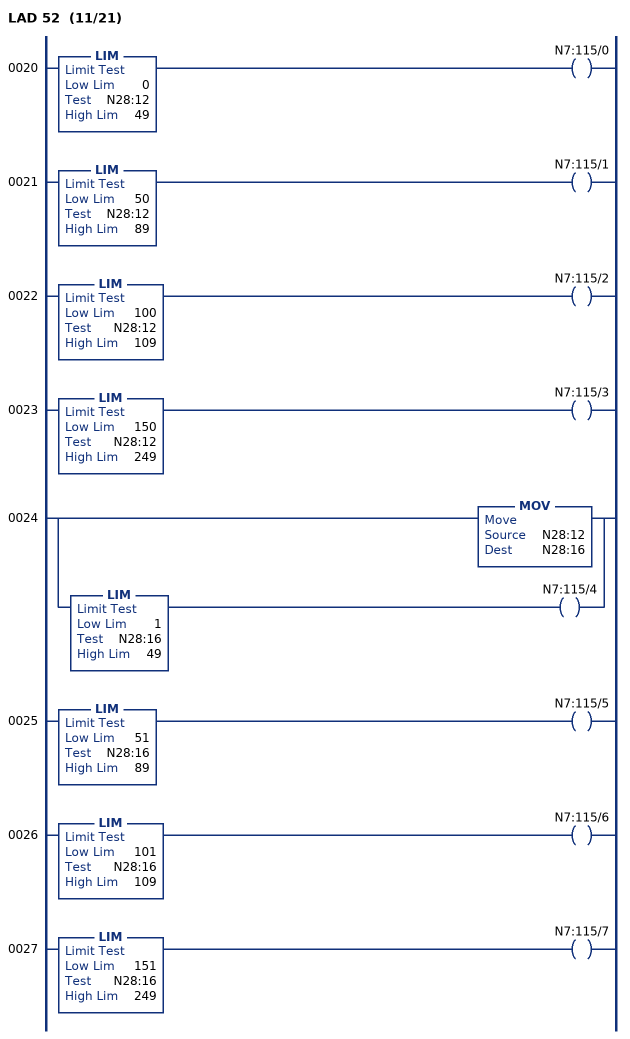
% Rung: 20 %
SOR LIM 0 N28:12 49 OTE N7:115/0 EOR
% Rung: 21 %
SOR LIM 50 N28:12 89 OTE N7:115/1 EOR
% Rung: 22 %
SOR LIM 100 N28:12 109 OTE N7:115/2 EOR
% Rung: 23 %
SOR LIM 150 N28:12 249 OTE N7:115/3 EOR
% Rung: 24 %
SOR BST MOV N28:12 N28:16 NXB LIM 1 N28:16 49 OTE N7:115/4 BND EOR
% Rung: 25 %
SOR LIM 51 N28:16 89 OTE N7:115/5 EOR
% Rung: 26 %
SOR LIM 101 N28:16 109 OTE N7:115/6 EOR
% Rung: 27 %
SOR LIM 151 N28:16 249 OTE N7:115/7 EOR

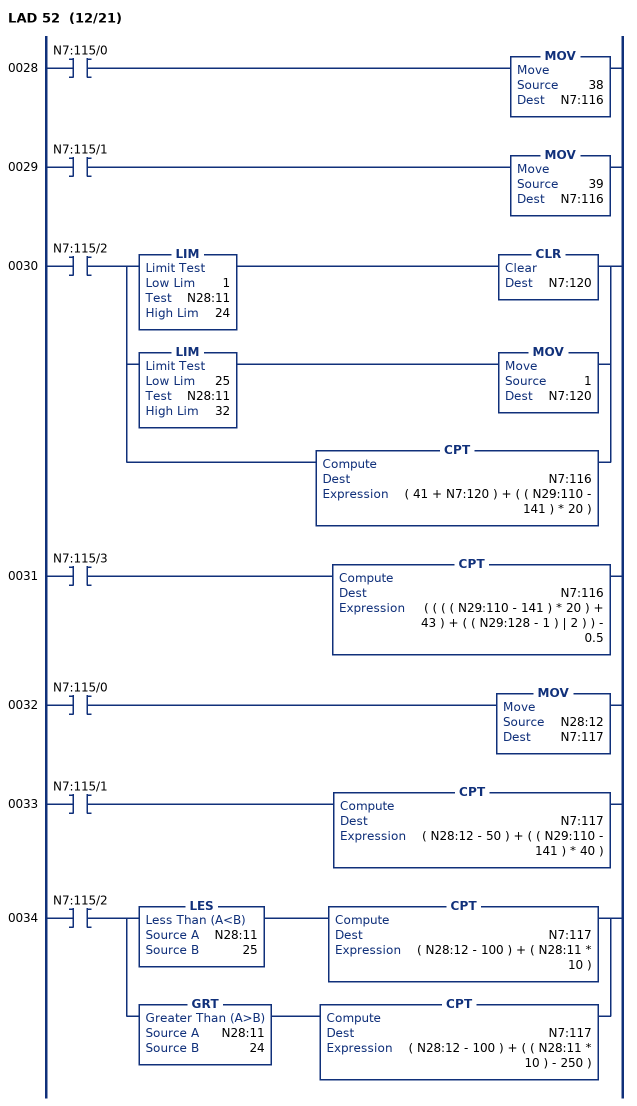
% Rung: 28 %
SOR XIC N7:115/0 MOV 38 N7:116 EOR
% Rung: 29 %
SOR XIC N7:115/1 MOV 39 N7:116 EOR
% Rung: 30 %
SOR XIC N7:115/2 BST LIM 1 N28:11 24 CLR N7:120 NXB LIM 25 N28:11 32 MOV 1 N7:120 NXB CPT N7:116 " ( 41 + N7:120 ) + ( ( N29:110 - 141 ) * 20 ) " BND EOR
% Rung: 31 %
SOR XIC N7:115/3 CPT N7:116 " ( ( ( ( N29:110 - 141 ) * 20 ) + 43 ) + ( ( N29:128 - 1 ) | 2 ) ) - 0.5 " EOR
% Rung: 32 %
SOR XIC N7:115/0 MOV N28:12 N7:117 EOR
% Rung: 33 %
SOR XIC N7:115/1 CPT N7:117 " ( N28:12 - 50 ) + ( ( N29:110 - 141 ) * 40 ) " EOR
% Rung: 34 %
SOR XIC N7:115/2 BST LES N28:11 25 CPT N7:117 " ( N28:12 - 100 ) + ( N28:11 * 10 ) " NXB GRT N28:11 24 CPT N7:117 " ( N28:12 - 100 ) + ( ( N28:11 * 10 ) - 250 ) " BND EOR

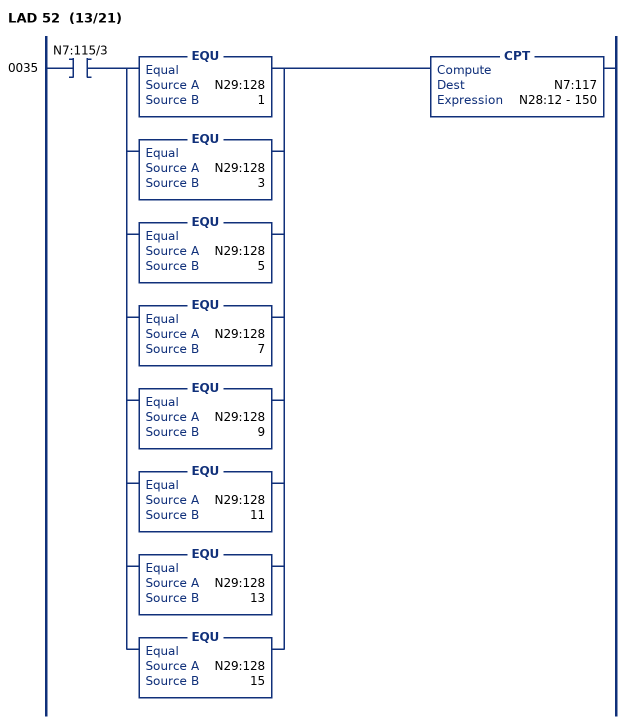
% Rung: 35 %
SOR XIC N7:115/3 BST EQU N29:128 1 NXB EQU N29:128 3 NXB EQU N29:128 5 NXB EQU N29:128 7 NXB EQU N29:128 9 NXB EQU N29:128 11 NXB EQU N29:128 13 NXB EQU N29:128 15 BND CPT N7:117 " N28:12 - 150 " EOR

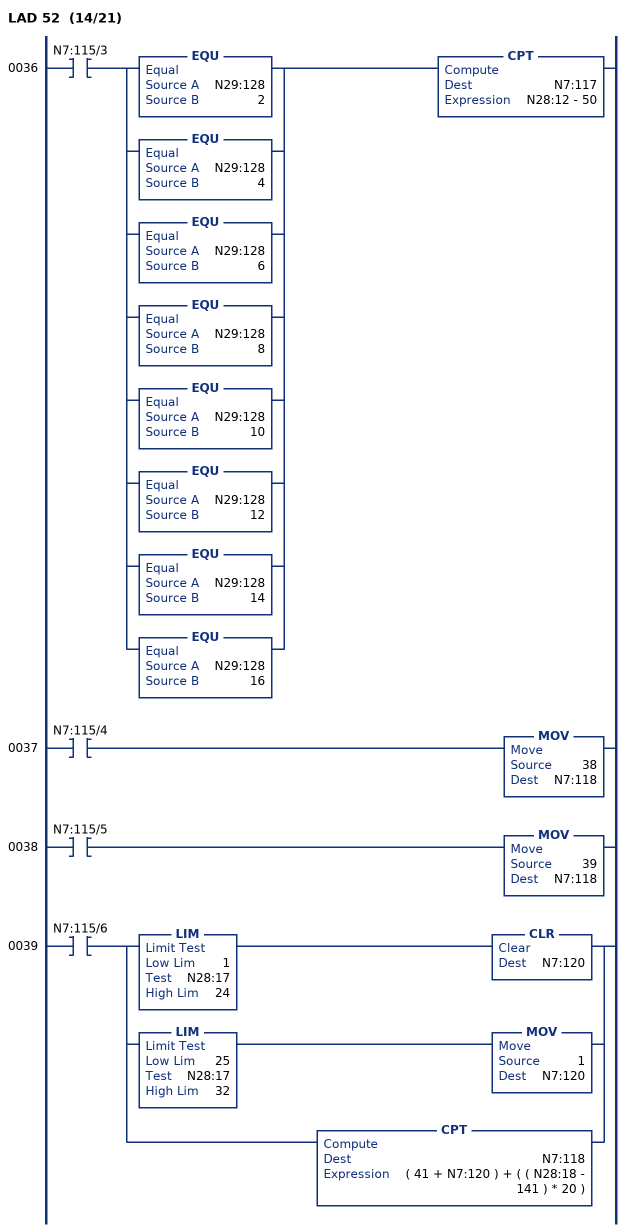
% Rung: 36 %
SOR XIC N7:115/3 BST EQU N29:128 2 NXB EQU N29:128 4 NXB EQU N29:128 6 NXB EQU N29:128 8 NXB EQU N29:128 10 NXB EQU N29:128 12 NXB EQU N29:128 14 NXB EQU N29:128 16 BND CPT N7:117 " N28:12 - 50 " EOR
% Rung: 37 %
SOR XIC N7:115/4 MOV 38 N7:118 EOR
% Rung: 38 %
SOR XIC N7:115/5 MOV 39 N7:118 EOR
% Rung: 39 %
SOR XIC N7:115/6 BST LIM 1 N28:17 24 CLR N7:120 NXB LIM 25 N28:17 32 MOV 1 N7:120 NXB CPT N7:118 " ( 41 + N7:120 ) + ( ( N28:18 - 141 ) * 20 ) " BND EOR

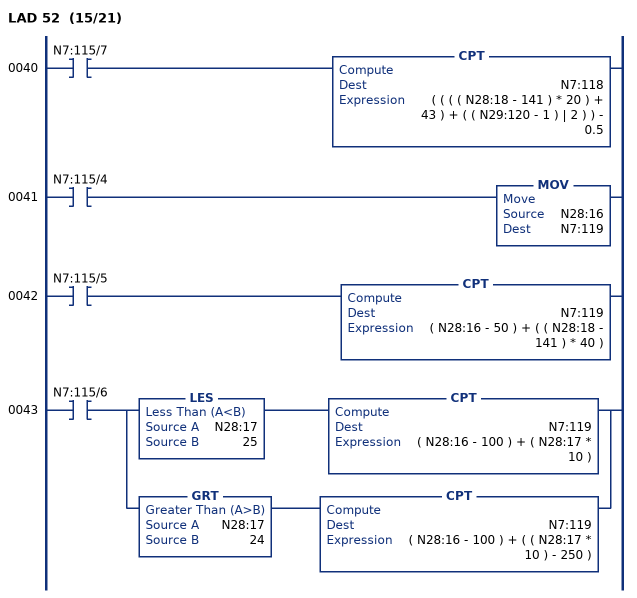
% Rung: 40 %
SOR XIC N7:115/7 CPT N7:118 " ( ( ( ( N28:18 - 141 ) * 20 ) + 43 ) + ( ( N29:120 - 1 ) | 2 ) ) - 0.5 " EOR
% Rung: 41 %
SOR XIC N7:115/4 MOV N28:16 N7:119 EOR
% Rung: 42 %
SOR XIC N7:115/5 CPT N7:119 " ( N28:16 - 50 ) + ( ( N28:18 - 141 ) * 40 ) " EOR
% Rung: 43 %
SOR XIC N7:115/6 BST LES N28:17 25 CPT N7:119 " ( N28:16 - 100 ) + ( N28:17 * 10 ) " NXB GRT N28:17 24 CPT N7:119 " ( N28:16 - 100 ) + ( ( N28:17 * 10 ) - 250 ) " BND EOR

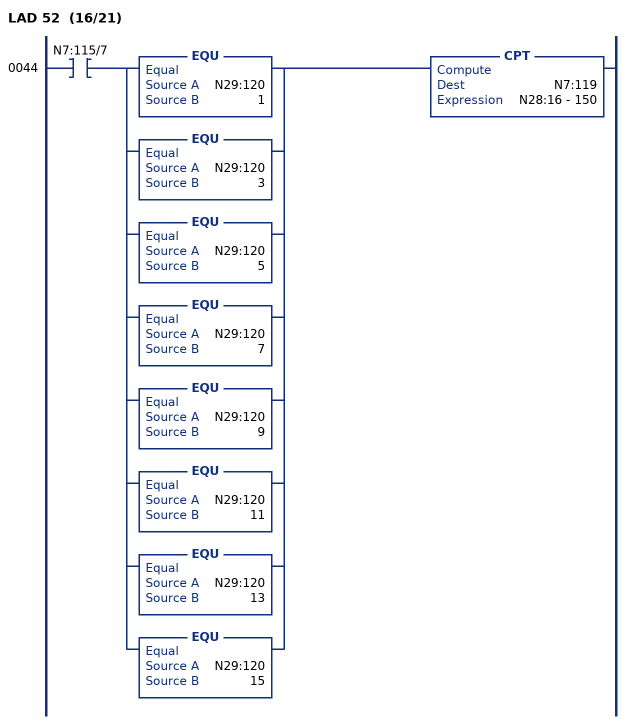
% Rung: 44 %
SOR XIC N7:115/7 BST EQU N29:120 1 NXB EQU N29:120 3 NXB EQU N29:120 5 NXB EQU N29:120 7 NXB EQU N29:120 9 NXB EQU N29:120 11 NXB EQU N29:120 13 NXB EQU N29:120 15 BND CPT N7:119 " N28:16 - 150 " EOR

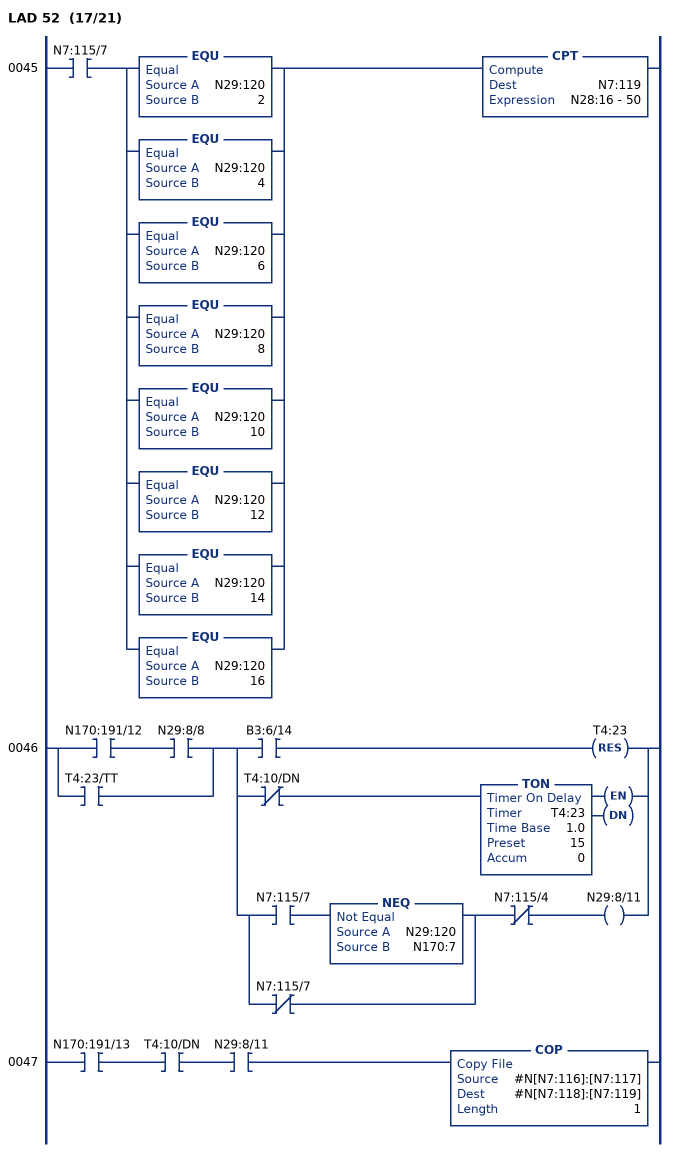
% Rung: 45 %
SOR XIC N7:115/7 BST EQU N29:120 2 NXB EQU N29:120 4 NXB EQU N29:120 6 NXB EQU N29:120 8 NXB EQU N29:120 10 NXB EQU N29:120 12 NXB EQU N29:120 14 NXB EQU N29:120 16 BND CPT N7:119 " N28:16 - 50 " EOR
% Rung: 46 %
SOR BST XIC N170:191/12 XIC N29:8/8 NXB XIC T4:23/TT BND BST XIC B3:6/14 RES T4:23 NXB XIO T4:10/DN TON T4:23 1.0 15 0 NXB BST XIC N7:115/7 NEQ N29:120 N170:7 NXB XIO N7:115/7 BND XIO N7:115/4 OTE N29:8/11 BND EOR
% Rung: 47 %
SOR XIC N170:191/13 XIC T4:10/DN XIC N29:8/11 COP #N[N7:116]:[N7:117] #N[N7:118]:[N7:119] 1 EOR

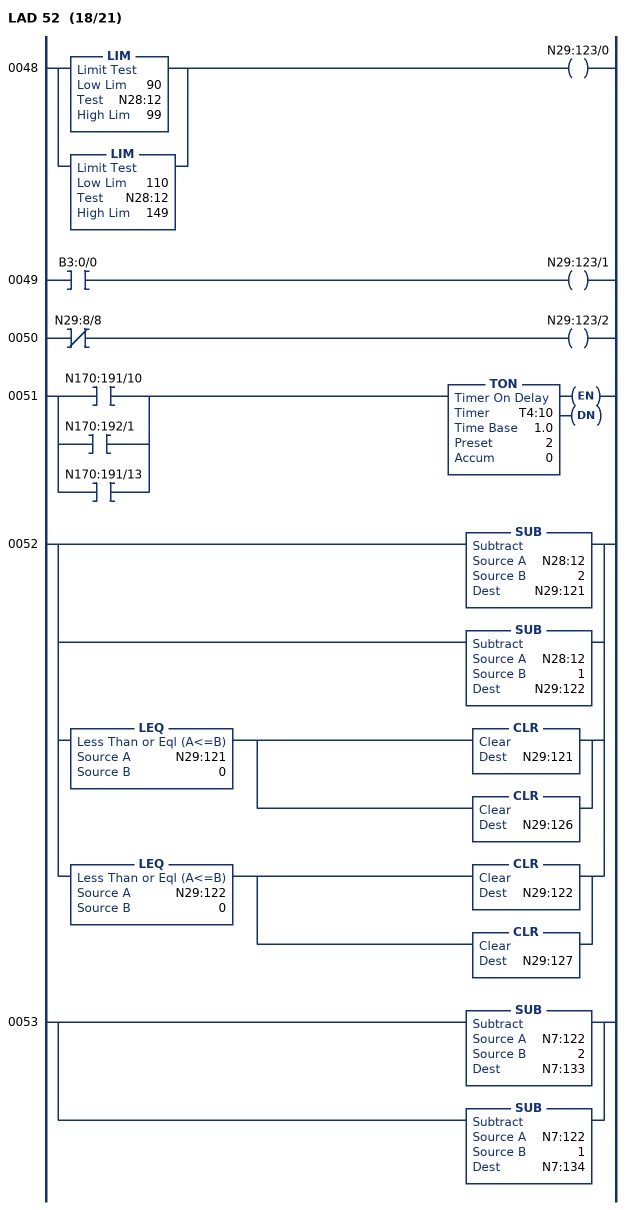
% Rung: 48 %
SOR BST LIM 90 N28:12 99 NXB LIM 110 N28:12 149 BND OTE N29:123/0 EOR
% Rung: 49 %
SOR XIC B3:0/0 OTE N29:123/1 EOR
% Rung: 50 %
SOR XIO N29:8/8 OTE N29:123/2 EOR
% Rung: 51 %
SOR BST XIC N170:191/10 NXB XIC N170:192/1 NXB XIC N170:191/13 BND TON T4:10 1.0 2 0 EOR
% Rung: 52 %
SOR BST SUB N28:12 2 N29:121 NXB SUB N28:12 1 N29:122 NXB LEQ N29:121 0 BST CLR N29:121 NXB CLR N29:126 BND NXB LEQ N29:122 0 BST CLR N29:122 NXB CLR N29:127 BND BND EOR
% Rung: 53 %
SOR BST SUB N7:122 2 N7:133 NXB SUB N7:122 1 N7:134 BND EOR

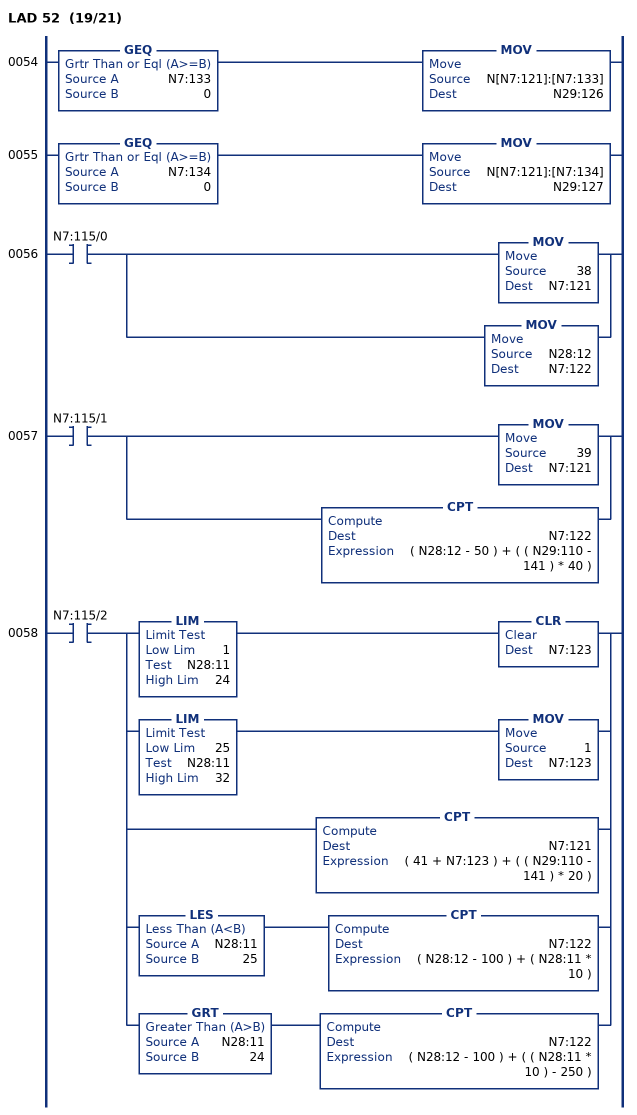
% Rung: 54 %
SOR GEQ N7:133 0 MOV N[N7:121]:[N7:133] N29:126 EOR
% Rung: 55 %
SOR GEQ N7:134 0 MOV N[N7:121]:[N7:134] N29:127 EOR
% Rung: 56 %
SOR XIC N7:115/0 BST MOV 38 N7:121 NXB MOV N28:12 N7:122 BND EOR
% Rung: 57 %
SOR XIC N7:115/1 BST MOV 39 N7:121 NXB CPT N7:122 " ( N28:12 - 50 ) + ( ( N29:110 - 141 ) * 40 ) " BND EOR
% Rung: 58 %
SOR XIC N7:115/2 BST LIM 1 N28:11 24 CLR N7:123 NXB LIM 25 N28:11 32 MOV 1 N7:123 NXB CPT N7:121 " ( 41 + N7:123 ) + ( ( N29:110 - 141 ) * 20 ) " NXB LES N28:11 25 CPT N7:122 " ( N28:12 - 100 ) + ( N28:11 * 10 ) " NXB GRT N28:11 24 CPT N7:122 " ( N28:12 - 100 ) + ( ( N28:11 * 10 ) - 250 ) " BND EOR

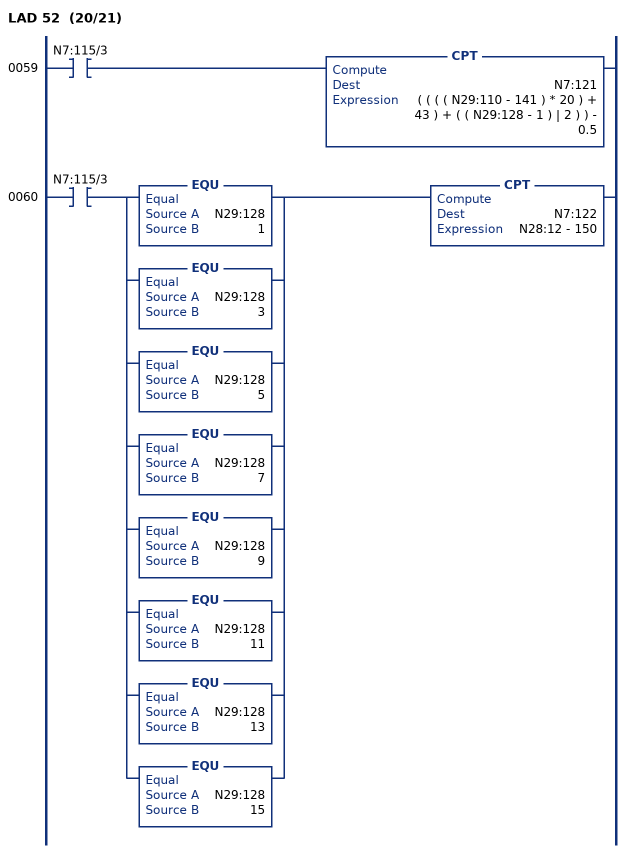
% Rung: 59 %
SOR XIC N7:115/3 CPT N7:121 " ( ( ( ( N29:110 - 141 ) * 20 ) + 43 ) + ( ( N29:128 - 1 ) | 2 ) ) - 0.5 " EOR
% Rung: 60 %
SOR XIC N7:115/3 BST EQU N29:128 1 NXB EQU N29:128 3 NXB EQU N29:128 5 NXB EQU N29:128 7 NXB EQU N29:128 9 NXB EQU N29:128 11 NXB EQU N29:128 13 NXB EQU N29:128 15 BND CPT N7:122 " N28:12 - 150 " EOR

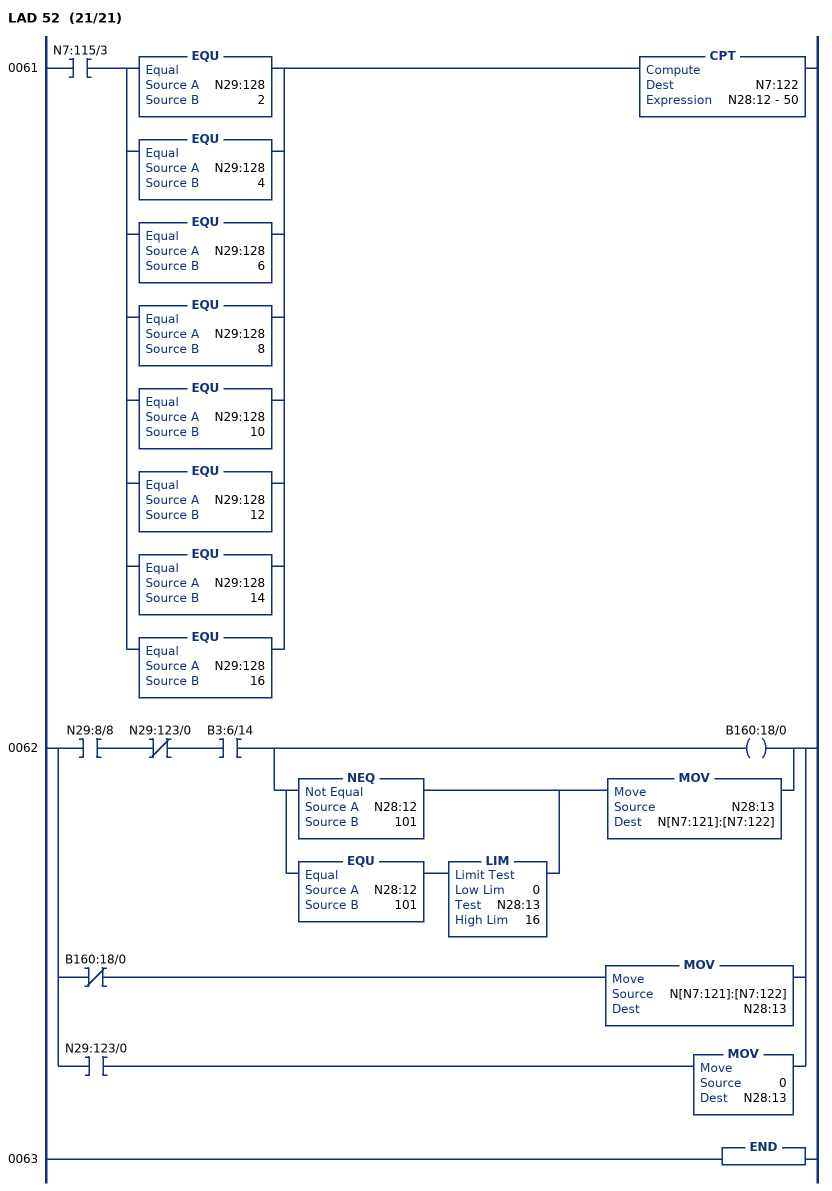
% Rung: 61 %
SOR XIC N7:115/3 BST EQU N29:128 2 NXB EQU N29:128 4 NXB EQU N29:128 6 NXB EQU N29:128 8 NXB EQU N29:128 10 NXB EQU N29:128 12 NXB EQU N29:128 14 NXB EQU N29:128 16 BND CPT N7:122 " N28:12 - 50 " EOR
% Rung: 62 %
SOR BST XIC N29:8/8 XIO N29:123/0 XIC B3:6/14 BST OTE B160:18/0 NXB BST NEQ N28:12 101 NXB EQU N28:12 101 LIM 0 N28:13 16 BND MOV N28:13 N[N7:121]:[N7:122] BND NXB XIO B160:18/0 MOV N[N7:121]:[N7:122] N28:13 NXB XIC N29:123/0 MOV 0 N28:13 BND EOR
% Rung: 63 %
SOR END EOR

LADDER 53
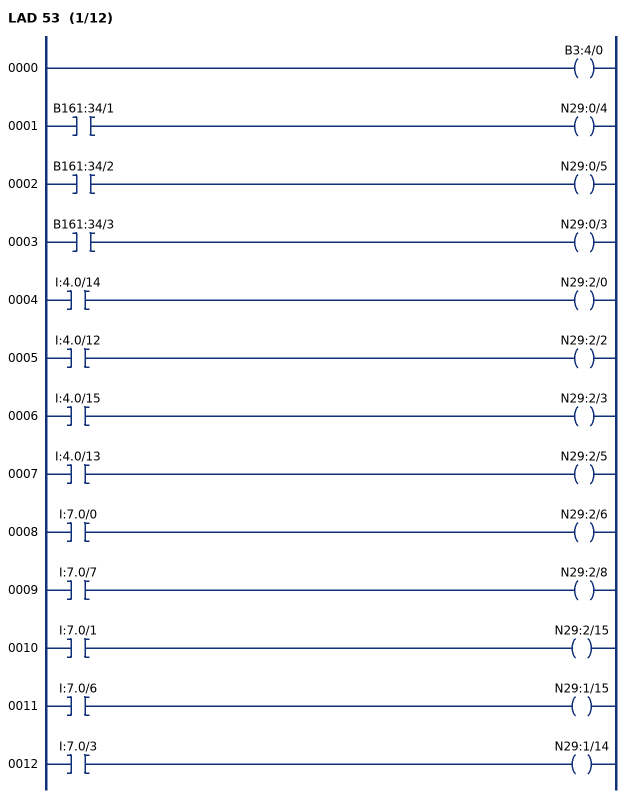
% Rung: 0 %
SOR OTE B3:4/0 EOR
% Rung: 1 %
SOR XIC B161:34/1 OTE N29:0/4 EOR
% Rung: 2 %
SOR XIC B161:34/2 OTE N29:0/5 EOR
% Rung: 3 %
SOR XIC B161:34/3 OTE N29:0/3 EOR
% Rung: 4 %
SOR XIC I:4.0/14 OTE N29:2/0 EOR
% Rung: 5 %
SOR XIC I:4.0/12 OTE N29:2/2 EOR
% Rung: 6 %
SOR XIC I:4.0/15 OTE N29:2/3 EOR
% Rung: 7 %
SOR XIC I:4.0/13 OTE N29:2/5 EOR
% Rung: 8 %
SOR XIC I:7.0/0 OTE N29:2/6 EOR
% Rung: 9 %
SOR XIC I:7.0/7 OTE N29:2/8 EOR
% Rung: 10 %
SOR XIC I:7.0/1 OTE N29:2/15 EOR
% Rung: 11 %
SOR XIC I:7.0/6 OTE N29:1/15 EOR
% Rung: 12 %
SOR XIC I:7.0/3 OTE N29:1/14 EOR

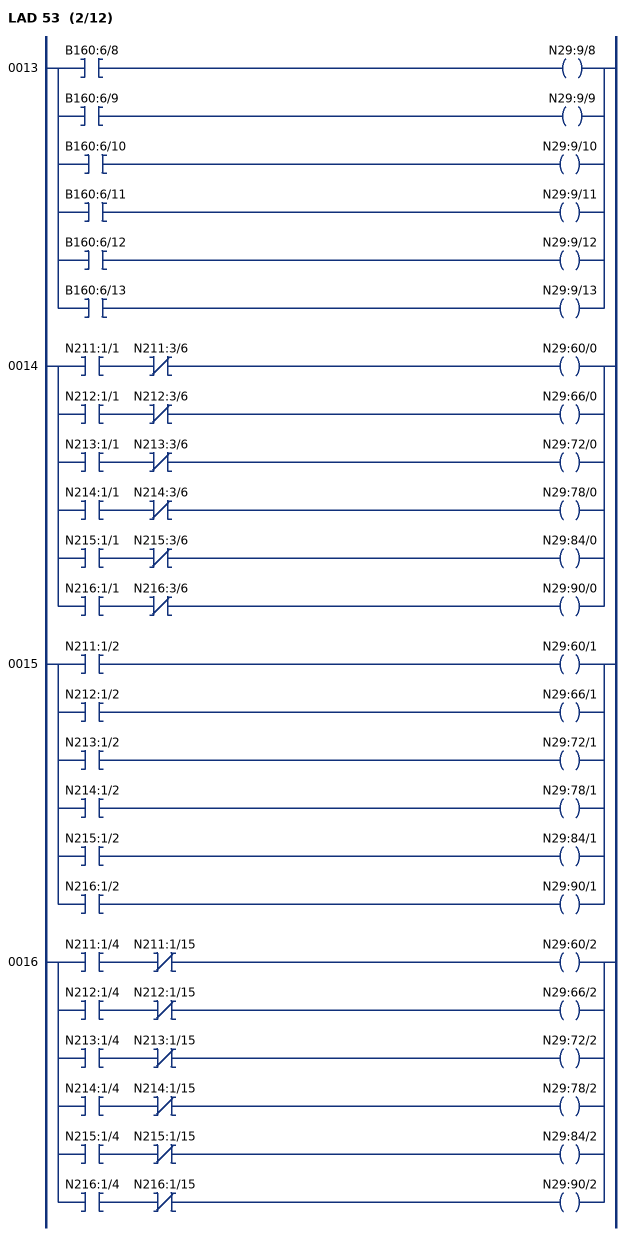
% Rung: 13 %
SOR BST XIC B160:6/8 OTE N29:9/8 NXB XIC B160:6/9 OTE N29:9/9 NXB XIC B160:6/10 OTE N29:9/10 NXB XIC B160:6/11 OTE N29:9/11 NXB XIC B160:6/12 OTE N29:9/12 NXB XIC B160:6/13 OTE N29:9/13 BND EOR
% Rung: 14 %
SOR BST XIC N211:1/1 XIO N211:3/6 OTE N29:60/0 NXB XIC N212:1/1 XIO N212:3/6 OTE N29:66/0 NXB XIC N213:1/1 XIO N213:3/6 OTE N29:72/0 NXB XIC N214:1/1 XIO N214:3/6 OTE N29:78/0 NXB XIC N215:1/1 XIO N215:3/6 OTE N29:84/0 NXB XIC N216:1/1 XIO N216:3/6 OTE N29:90/0 BND EOR
% Rung: 15 %
SOR BST XIC N211:1/2 OTE N29:60/1 NXB XIC N212:1/2 OTE N29:66/1 NXB XIC N213:1/2 OTE N29:72/1 NXB XIC N214:1/2 OTE N29:78/1 NXB XIC N215:1/2 OTE N29:84/1 NXB XIC N216:1/2 OTE N29:90/1 BND EOR
% Rung: 16 %
SOR BST XIC N211:1/4 XIO N211:1/15 OTE N29:60/2 NXB XIC N212:1/4 XIO N212:1/15 OTE N29:66/2 NXB XIC N213:1/4 XIO N213:1/15 OTE N29:72/2 NXB XIC N214:1/4 XIO N214:1/15 OTE N29:78/2 NXB XIC N215:1/4 XIO N215:1/15 OTE N29:84/2 NXB XIC N216:1/4 XIO N216:1/15 OTE N29:90/2 BND EOR

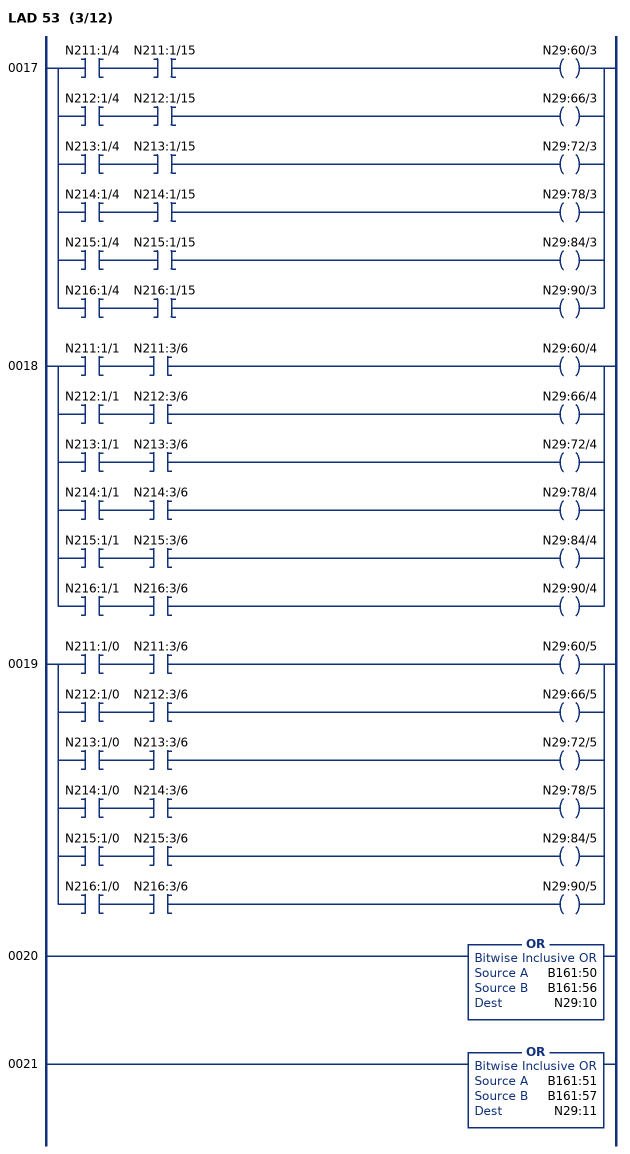
% Rung: 17 %
SOR BST XIC N211:1/4 XIC N211:1/15 OTE N29:60/3 NXB XIC N212:1/4 XIC N212:1/15 OTE N29:66/3 NXB XIC N213:1/4 XIC N213:1/15 OTE N29:72/3 NXB XIC N214:1/4 XIC N214:1/15 OTE N29:78/3 NXB XIC N215:1/4 XIC N215:1/15 OTE N29:84/3 NXB XIC N216:1/4 XIC N216:1/15 OTE N29:90/3 BND EOR
% Rung: 18 %
SOR BST XIC N211:1/1 XIC N211:3/6 OTE N29:60/4 NXB XIC N212:1/1 XIC N212:3/6 OTE N29:66/4 NXB XIC N213:1/1 XIC N213:3/6 OTE N29:72/4 NXB XIC N214:1/1 XIC N214:3/6 OTE N29:78/4 NXB XIC N215:1/1 XIC N215:3/6 OTE N29:84/4 NXB XIC N216:1/1 XIC N216:3/6 OTE N29:90/4 BND EOR
% Rung: 19 %
SOR BST XIC N211:1/0 XIC N211:3/6 OTE N29:60/5 NXB XIC N212:1/0 XIC N212:3/6 OTE N29:66/5 NXB XIC N213:1/0 XIC N213:3/6 OTE N29:72/5 NXB XIC N214:1/0 XIC N214:3/6 OTE N29:78/5 NXB XIC N215:1/0 XIC N215:3/6 OTE N29:84/5 NXB XIC N216:1/0 XIC N216:3/6 OTE N29:90/5 BND EOR
% Rung: 20 %
SOR OR B161:50 B161:56 N29:10 EOR
% Rung: 21 %
SOR OR B161:51 B161:57 N29:11 EOR

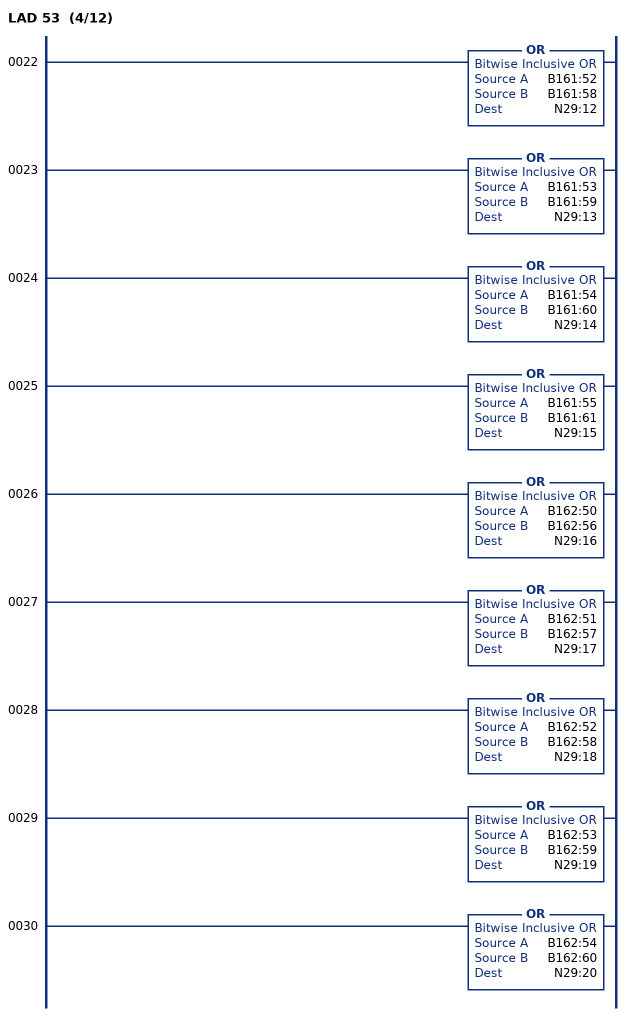
% Rung: 22 %
SOR OR B161:52 B161:58 N29:12 EOR
% Rung: 23 %
SOR OR B161:53 B161:59 N29:13 EOR
% Rung: 24 %
SOR OR B161:54 B161:60 N29:14 EOR
% Rung: 25 %
SOR OR B161:55 B161:61 N29:15 EOR
% Rung: 26 %
SOR OR B162:50 B162:56 N29:16 EOR
% Rung: 27 %
SOR OR B162:51 B162:57 N29:17 EOR
% Rung: 28 %
SOR OR B162:52 B162:58 N29:18 EOR
% Rung: 29 %
SOR OR B162:53 B162:59 N29:19 EOR
% Rung: 30 %
SOR OR B162:54 B162:60 N29:20 EOR

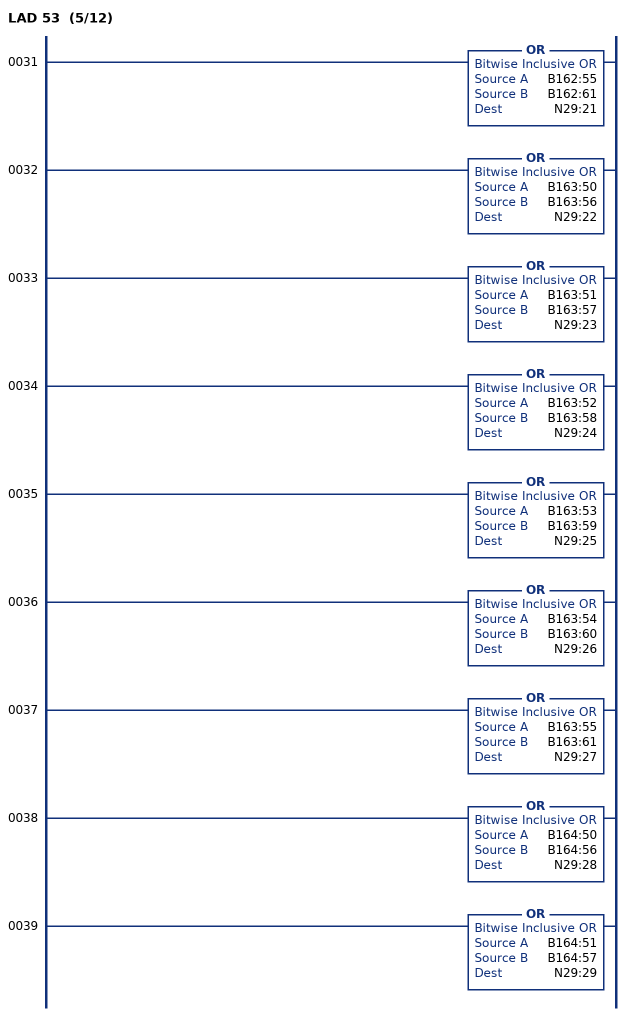
% Rung: 31 %
SOR OR B162:55 B162:61 N29:21 EOR
% Rung: 32 %
SOR OR B163:50 B163:56 N29:22 EOR
% Rung: 33 %
SOR OR B163:51 B163:57 N29:23 EOR
% Rung: 34 %
SOR OR B163:52 B163:58 N29:24 EOR
% Rung: 35 %
SOR OR B163:53 B163:59 N29:25 EOR
% Rung: 36 %
SOR OR B163:54 B163:60 N29:26 EOR
% Rung: 37 %
SOR OR B163:55 B163:61 N29:27 EOR
% Rung: 38 %
SOR OR B164:50 B164:56 N29:28 EOR
% Rung: 39 %
SOR OR B164:51 B164:57 N29:29 EOR

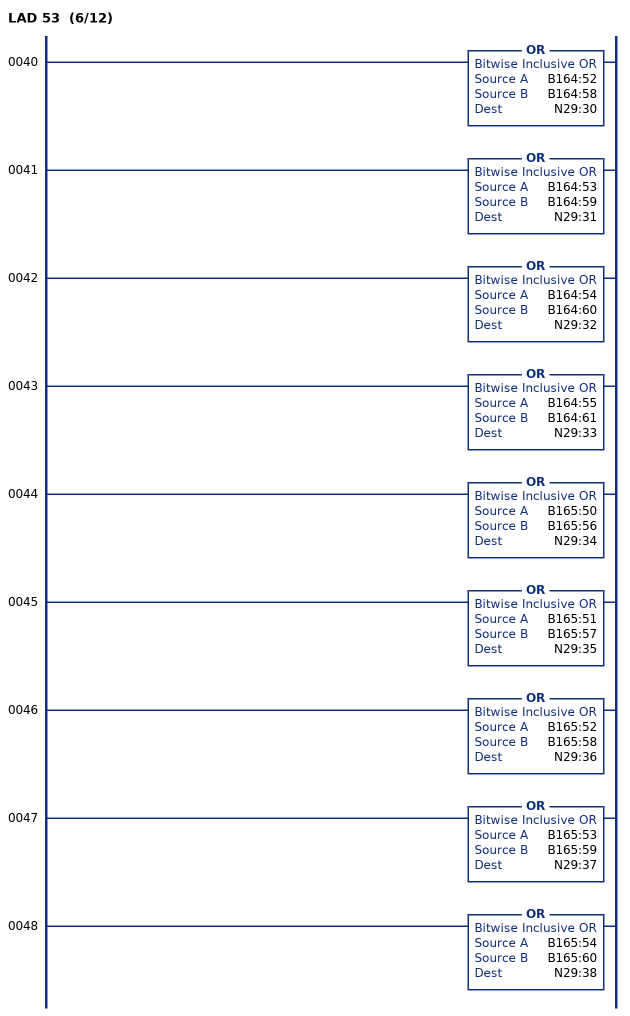
% Rung: 40 %
SOR OR B164:52 B164:58 N29:30 EOR
% Rung: 41 %
SOR OR B164:53 B164:59 N29:31 EOR
% Rung: 42 %
SOR OR B164:54 B164:60 N29:32 EOR
% Rung: 43 %
SOR OR B164:55 B164:61 N29:33 EOR
% Rung: 44 %
SOR OR B165:50 B165:56 N29:34 EOR
% Rung: 45 %
SOR OR B165:51 B165:57 N29:35 EOR
% Rung: 46 %
SOR OR B165:52 B165:58 N29:36 EOR
% Rung: 47 %
SOR OR B165:53 B165:59 N29:37 EOR
% Rung: 48 %
SOR OR B165:54 B165:60 N29:38 EOR

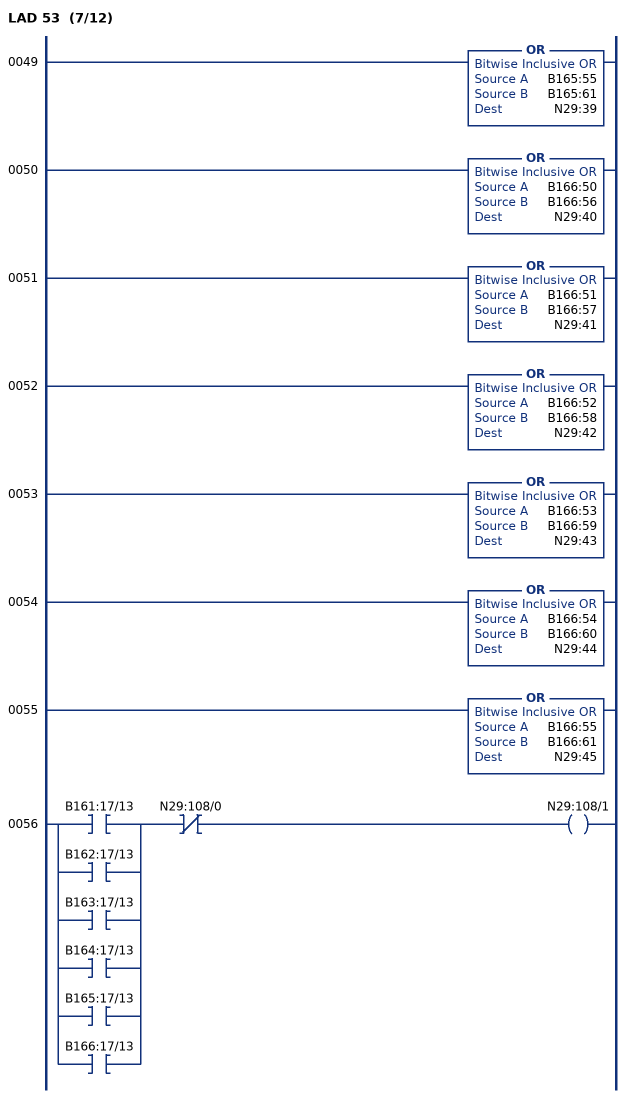
% Rung: 49 %
SOR OR B165:55 B165:61 N29:39 EOR
% Rung: 50 %
SOR OR B166:50 B166:56 N29:40 EOR
% Rung: 51 %
SOR OR B166:51 B166:57 N29:41 EOR
% Rung: 52 %
SOR OR B166:52 B166:58 N29:42 EOR
% Rung: 53 %
SOR OR B166:53 B166:59 N29:43 EOR
% Rung: 54 %
SOR OR B166:54 B166:60 N29:44 EOR
% Rung: 55 %
SOR OR B166:55 B166:61 N29:45 EOR
% Rung: 56 %
SOR BST XIC B161:17/13 NXB XIC B162:17/13 NXB XIC B163:17/13 NXB XIC B164:17/13 NXB XIC B165:17/13 NXB XIC B166:17/13 BND XIO N29:108/0 OTE N29:108/1 EOR

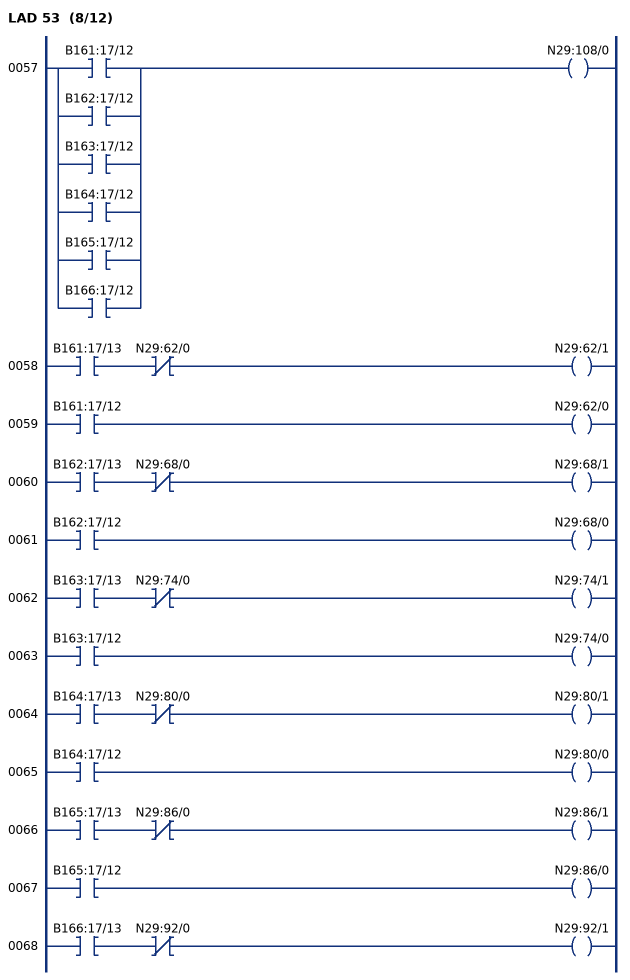
% Rung: 57 %
SOR BST XIC B161:17/12 NXB XIC B162:17/12 NXB XIC B163:17/12 NXB XIC B164:17/12 NXB XIC B165:17/12 NXB XIC B166:17/12 BND OTE N29:108/0 EOR
% Rung: 58 %
SOR XIC B161:17/13 XIO N29:62/0 OTE N29:62/1 EOR
% Rung: 59 %
SOR XIC B161:17/12 OTE N29:62/0 EOR
% Rung: 60 %
SOR XIC B162:17/13 XIO N29:68/0 OTE N29:68/1 EOR
% Rung: 61 %
SOR XIC B162:17/12 OTE N29:68/0 EOR
% Rung: 62 %
SOR XIC B163:17/13 XIO N29:74/0 OTE N29:74/1 EOR
% Rung: 63 %
SOR XIC B163:17/12 OTE N29:74/0 EOR
% Rung: 64 %
SOR XIC B164:17/13 XIO N29:80/0 OTE N29:80/1 EOR
% Rung: 65 %
SOR XIC B164:17/12 OTE N29:80/0 EOR
% Rung: 66 %
SOR XIC B165:17/13 XIO N29:86/0 OTE N29:86/1 EOR
% Rung: 67 %
SOR XIC B165:17/12 OTE N29:86/0 EOR
% Rung: 68 %
SOR XIC B166:17/13 XIO N29:92/0 OTE N29:92/1 EOR

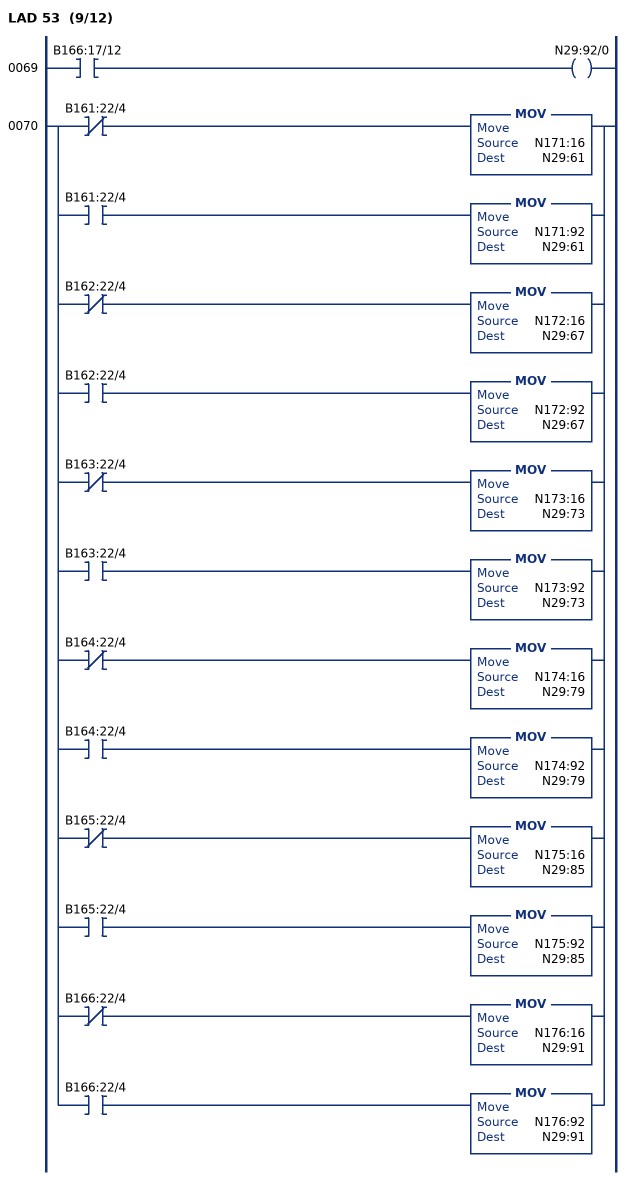
% Rung: 69 %
SOR XIC B166:17/12 OTE N29:92/0 EOR
% Rung: 70 %
SOR BST BST XIO B161:22/4 MOV N171:16 N29:61 NXB XIC B161:22/4 MOV N171:92 N29:61 BND NXB BST XIO B162:22/4 MOV N172:16 N29:67 NXB XIC B162:22/4 MOV N172:92 N29:67 BND NXB BST XIO B163:22/4 MOV N173:16 N29:73 NXB XIC B163:22/4 MOV N173:92 N29:73 BND NXB BST XIO B164:22/4 MOV N174:16 N29:79 NXB XIC B164:22/4 MOV N174:92 N29:79 BND NXB BST XIO B165:22/4 MOV N175:16 N29:85 NXB XIC B165:22/4 MOV N175:92 N29:85 BND NXB BST XIO B166:22/4 MOV N176:16 N29:91 NXB XIC B166:22/4 MOV N176:92 N29:91 BND BND EOR

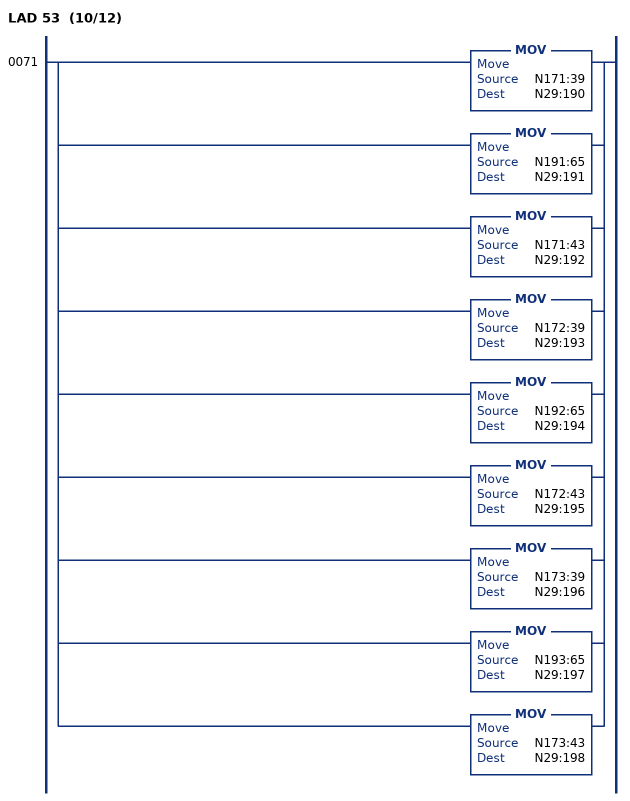
% Rung: 71 %
SOR BST BST BST MOV N171:39 N29:190 NXB MOV N191:65 N29:191 NXB MOV N171:43 N29:192 BND NXB MOV N172:39 N29:193 NXB MOV N192:65 N29:194 NXB MOV N172:43 N29:195 BND NXB MOV N173:39 N29:196 NXB MOV N193:65 N29:197 NXB MOV N173:43 N29:198 BND EOR

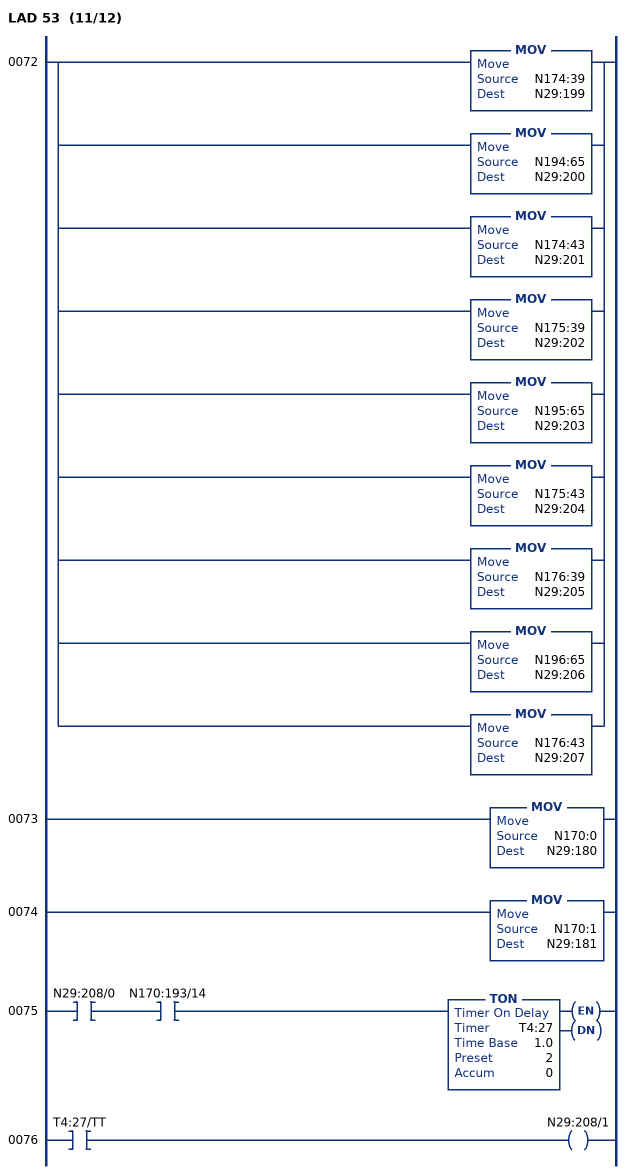
% Rung: 72 %
SOR BST BST BST MOV N174:39 N29:199 NXB MOV N194:65 N29:200 NXB MOV N174:43 N29:201 BND NXB MOV N175:39 N29:202 NXB MOV N195:65 N29:203 NXB MOV N175:43 N29:204 BND NXB MOV N176:39 N29:205 NXB MOV N196:65 N29:206 NXB MOV N176:43 N29:207 BND EOR
% Rung: 73 %
SOR MOV N170:0 N29:180 EOR
% Rung: 74 %
SOR MOV N170:1 N29:181 EOR
% Rung: 75 %
SOR XIC N29:208/0 XIC N170:193/14 TON T4:27 1.0 2 0 EOR
% Rung: 76 %
SOR XIC T4:27/TT OTE N29:208/1 EOR

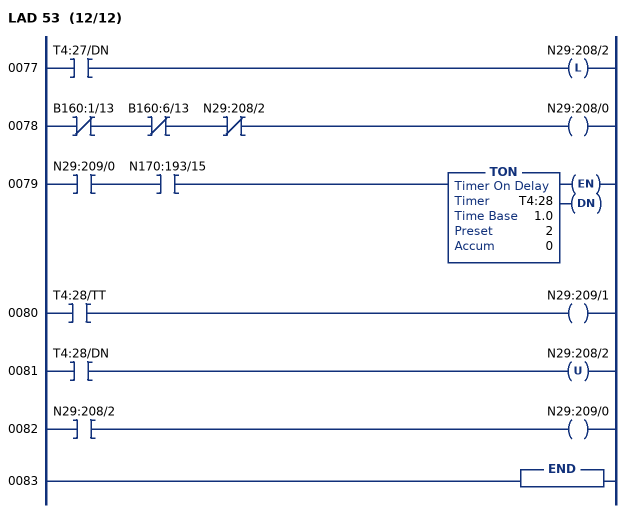
% Rung: 77 %
SOR XIC T4:27/DN OTL N29:208/2 EOR
% Rung: 78 %
SOR XIO B160:1/13 XIO B160:6/13 XIO N29:208/2 OTE N29:208/0 EOR
% Rung: 79 %
SOR XIC N29:209/0 XIC N170:193/15 TON T4:28 1.0 2 0 EOR
% Rung: 80 %
SOR XIC T4:28/TT OTE N29:209/1 EOR
% Rung: 81 %
SOR XIC T4:28/DN OTU N29:208/2 EOR
% Rung: 82 %
SOR XIC N29:208/2 OTE N29:209/0 EOR
% Rung: 83 %
SOR END EOR

LADDER 71
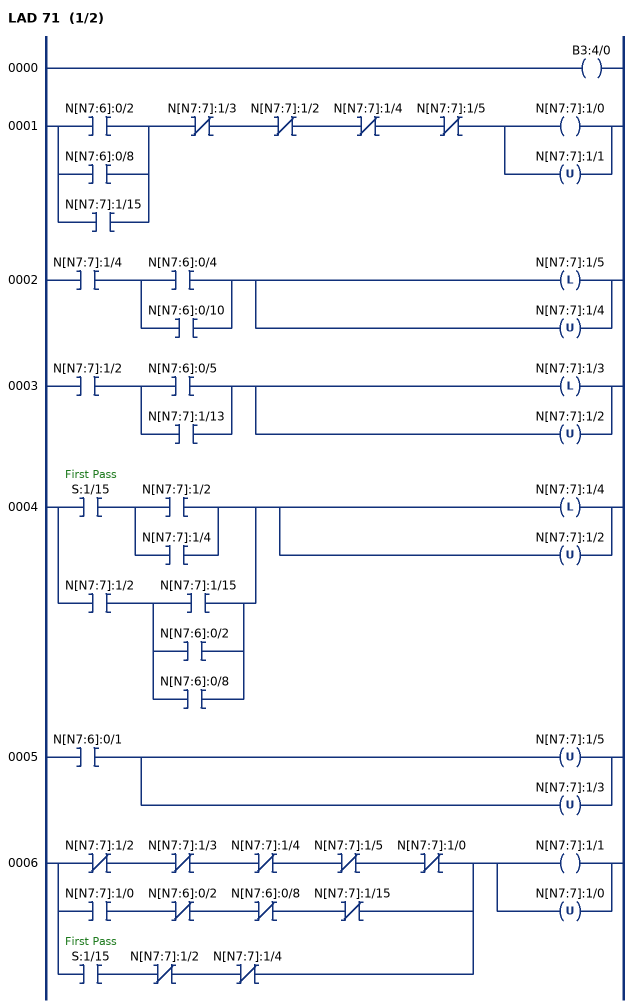
% Rung: 0 %
SOR OTE B3:4/0 EOR
% Rung: 1 %
SOR BST XIC N[N7:6]:0/2 NXB XIC N[N7:6]:0/8 NXB XIC N[N7:7]:1/15 BND XIO N[N7:7]:1/3 XIO N[N7:7]:1/2 XIO N[N7:7]:1/4 XIO N[N7:7]:1/5 BST OTE N[N7:7]:1/0 NXB OTU N[N7:7]:1/1 BND EOR
% Rung: 2 %
SOR XIC N[N7:7]:1/4 BST XIC N[N7:6]:0/4 NXB XIC N[N7:6]:0/10 BND BST OTL N[N7:7]:1/5 NXB OTU N[N7:7]:1/4 BND EOR
% Rung: 3 %
SOR XIC N[N7:7]:1/2 BST XIC N[N7:6]:0/5 NXB XIC N[N7:7]:1/13 BND BST OTL N[N7:7]:1/3 NXB OTU N[N7:7]:1/2 BND EOR
% Rung: 4 %
SOR BST XIC S:1/15 BST XIC N[N7:7]:1/2 NXB XIC N[N7:7]:1/4 BND NXB XIC N[N7:7]:1/2 BST XIC N[N7:7]:1/15 NXB XIC N[N7:6]:0/2 NXB XIC N[N7:6]:0/8 BND BND BST OTL N[N7:7]:1/4 NXB OTU N[N7:7]:1/2 BND EOR
%   S:1/15  "First Pass" %
% Rung: 5 %
SOR XIC N[N7:6]:0/1 BST OTU N[N7:7]:1/5 NXB OTU N[N7:7]:1/3 BND EOR
% Rung: 6 %
SOR BST XIO N[N7:7]:1/2 XIO N[N7:7]:1/3 XIO N[N7:7]:1/4 XIO N[N7:7]:1/5 XIO N[N7:7]:1/0 NXB XIC N[N7:7]:1/0 XIO N[N7:6]:0/2 XIO N[N7:6]:0/8 XIO N[N7:7]:1/15 NXB XIC S:1/15 XIO N[N7:7]:1/2 XIO N[N7:7]:1/4 BND BST OTE N[N7:7]:1/1 NXB OTU N[N7:7]:1/0 BND EOR
%   S:1/15  "First Pass" %

